// TIA Portal V17 export
// export: Created 2023-07-20T16:54:10.2043387Z, ExportSetting WithDefaults, DisplayName Totally Integrated Automation Portal, DisplayVersion V17, DisplayName TIA Portal Openness, DisplayVersion V17, DisplayName TIA Portal Version Control Interface, DisplayVersion V17, DisplayName STEP 7 Professional, DisplayVersion V17, DisplayName STEP 7 Safety, DisplayVersion V17, DisplayName WinCC Professional, DisplayVersion V17
DATA_BLOCK "Modbus RTU RW sequencer_DB"   // DB5002
VERSION : 0.1
// stored: AutoNumber false, DBAccessibleFromOPCUA true, InstanceOfName Modbus RTU RW sequencer, InstanceOfType FB
"Modbus RTU RW sequencer"
   // VAR
   //    "Operation data number" { S7_SetPoint := 'True'} : "Deconcatenate UDInt into two UInt";
   //    "Operation type" { S7_SetPoint := 'True'} : "Deconcatenate UDInt into two UInt";
   //    Position { S7_SetPoint := 'True'} : "Deconcatenate UDInt into two UInt";
   //    Speed { S7_SetPoint := 'True'} : "Deconcatenate UDInt into two UInt";
   //    "Starting changing rate" { S7_SetPoint := 'True'} : "Deconcatenate UDInt into two UInt";
   //    "Stopping deceleration" { S7_SetPoint := 'True'} : "Deconcatenate UDInt into two UInt";
   //    "Operating current" { S7_SetPoint := 'True'} : "Deconcatenate UDInt into two UInt";
   //    "Operation trigger" { S7_SetPoint := 'True'} : "Deconcatenate UDInt into two UInt";
   //    "Forwarding destination" { S7_SetPoint := 'True'} : "Deconcatenate UDInt into two UInt";
   //    "Alarm reset" { S7_SetPoint := 'True'} : "Deconcatenate UDInt into two UInt";
   //    "Clear alarm history" { S7_SetPoint := 'True'} : "Deconcatenate UDInt into two UInt";
   //    "Clear comm history" { S7_SetPoint := 'True'} : "Deconcatenate UDInt into two UInt";
   //    "Clear monitor alarm history" { S7_SetPoint := 'True'} : "Deconcatenate UDInt into two UInt";
   //    "Clear comm history_1" { S7_SetPoint := 'True'} : "Deconcatenate UDInt into two UInt";
   //    "Monitor present alarm" { S7_SetPoint := 'True'} : "Concatenate two UInt into one UDInt";
   //    "Monitor alarm history 1" { S7_SetPoint := 'True'} : "Concatenate two UInt into one UDInt";
   //    "Monitor alarm history 2" { S7_SetPoint := 'True'} : "Concatenate two UInt into one UDInt";
   //    "Monitor alarm history 3" { S7_SetPoint := 'True'} : "Concatenate two UInt into one UDInt";
   //    "Monitor alarm history 4" { S7_SetPoint := 'True'} : "Concatenate two UInt into one UDInt";
   //    "Monitor alarm history 5" { S7_SetPoint := 'True'} : "Concatenate two UInt into one UDInt";
   //    "Monitor present communication error" { S7_SetPoint := 'True'} : "Concatenate two UInt into one UDInt";
   //    "Monitor communication error history 1" { S7_SetPoint := 'True'} : "Concatenate two UInt into one UDInt";
   //    "Monitor communication error history 2" { S7_SetPoint := 'True'} : "Concatenate two UInt into one UDInt";
   //    "Monitor communication error history 3" { S7_SetPoint := 'True'} : "Concatenate two UInt into one UDInt";
   //    "Monitor communication error history 4" { S7_SetPoint := 'True'} : "Concatenate two UInt into one UDInt";
   //    "Monitor communication error history 5" { S7_SetPoint := 'True'} : "Concatenate two UInt into one UDInt";
   //    "Monitor feedback position" { S7_SetPoint := 'True'} : "Concatenate two UInt into one UDInt";
   //    "Monitor feedback speed r/min" { S7_SetPoint := 'True'} : "Concatenate two UInt into one UDInt";
   //    "Monitor feedback speed Hz" { S7_SetPoint := 'True'} : "Concatenate two UInt into one UDInt";
   //    "Monitor direct I/O" { S7_SetPoint := 'True'} : "Concatenate two UInt into one UDInt";
   //    "Monitor torque" { S7_SetPoint := 'True'} : "Concatenate two UInt into one UDInt";
   //    "Monitor cumulative load" { S7_SetPoint := 'True'} : "Concatenate two UInt into one UDInt";
   //    "Monitor driver temperature" { S7_SetPoint := 'True'} : "Concatenate two UInt into one UDInt";
   //    "Monitor motor temperature" { S7_SetPoint := 'True'} : "Concatenate two UInt into one UDInt";
   //    "Monitor inverter voltage" { S7_SetPoint := 'True'} : "Concatenate two UInt into one UDInt";
   //    "Monitor power supply voltage" { S7_SetPoint := 'True'} : "Concatenate two UInt into one UDInt";
   //    "Monitor DIP SW" { S7_SetPoint := 'True'} : "Concatenate two UInt into one UDInt";
   //    "Monitor ROT SW0" { S7_SetPoint := 'True'} : "Concatenate two UInt into one UDInt";
   //    "Monitor ROT SW1" { S7_SetPoint := 'True'} : "Concatenate two UInt into one UDInt";
   // END_VAR
BEGIN
END_DATA_BLOCK
